//********************************Action case***********************************
CASE fb_mem.STS.State OF
	E_State_PackML.IDLE 			: 
		//Do nothing
	E_State_PackML.STARTING 		:
		Motor.Start();
		IF Motor.State = E_State_PackML.EXECUTE THEN
			fb_mem.STS.Starting_SC 		:= TRUE;	
		END_IF
	E_State_PackML.EXECUTE 			: 
		//Do nothing
	E_State_PackML.COMPLETING		:
		Motor.Stop();
		fb_mem.STS.Completing_SC := TRUE;
	E_State_PackML.COMPLETE 		:
		//Do nothing
	E_State_PackML.RESETTING 		:
		Motor.Reset();
		IF Motor.State = E_State_PackML.IDLE THEN
			fb_mem.STS.Resetting_SC 	:= TRUE;
		END_IF
	E_State_PackML.HOLDING 			:
		Motor.Stop();
		IF Motor.State = E_State_PackML.STOPPED THEN
			fb_mem.STS.Holding_SC		:= TRUE;
		END_IF
	E_State_PackML.HELD 			:
		//Do nothing
	E_State_PackML.UNHOLDING 		:
		Motor.Reset();
		Motor.Reset();
		IF Motor.State = E_State_PackML.EXECUTE THEN
			fb_mem.STS.Unholding_SC		:= TRUE;
		END_IF
	E_State_PackML.SUSPENDING 		:
		Motor.Stop();
		IF Motor.State = E_State_PackML.STOPPED THEN
			fb_mem.STS.Suspending_SC 	:= TRUE;
		END_IF
	E_State_PackML.SUSPENDED 		:
		//Do nothing
	E_State_PackML.UNSUSPENDING 	:
		Motor.Reset();
		Motor.Reset();
		IF Motor.State = E_State_PackML.EXECUTE THEN
			fb_mem.CS.Unsuspend 		:= TRUE;
		END_IF
	E_State_PackML.ABORTING			:
		Motor.Abort();
		IF Motor.State = E_State_PackML.ABORTED THEN
			fb_mem.STS.Aborting_SC 		:= TRUE;
		END_IF
	E_State_PackML.ABORTED			:		
		//Do nothing
	E_State_PackML.CLEARING 		:
		Motor.Clear();
		IF Motor.State = E_State_PackML.STOPPED THEN
			fb_mem.STS.Clearing_SC 		:= TRUE;
		END_IF
	E_State_PackML.STOPPING 		:
		IF Motor.State = E_State_PackML.STOPPED THEN
			fb_mem.STS.Stopping_SC 		:= TRUE;
		END_IF
	E_State_PackML.STOPPED 			:
		//Do nothing
END_CASE

//********************************HMI_Connection***********************************
fb_mem.STS.StringState     := TO_STRING(fb_mem.STS.State); 

//********************************ZEROING***********************************

fb_mem.CS.Auto            := FALSE;
fb_mem.CS.Manueel         := FALSE;
fb_mem.CS.Start           := FALSE;
fb_mem.CS.Stop            := FALSE;
fb_mem.CS.Reset           := FALSE;
fb_mem.CS.Abort           := FALSE;
fb_mem.CS.Clear           := FALSE;
fb_mem.CS.UnSuspend       := FALSE;
fb_mem.CS.Suspend         := FALSE;
fb_mem.CS.UnHold          := FALSE;
fb_mem.CS.Hold            := FALSE;

{warning 'add method implementation '}
METHOD Abort : BOOL
fb_mem.CS.Abort := TRUE;
END_METHOD

METHOD Aborting_SC : BOOL
VAR_INPUT
END_VAR
fb_mem.STS.Aborting_SC := TRUE;
END_METHOD

{warning 'add method implementation '}
METHOD Auto : BOOL
fb_mem.CS.Auto := TRUE;
Auto := fb_mem.STS.Auto;
END_METHOD

{warning 'add method implementation '}
METHOD Clear : BOOL
fb_mem.CS.Clear := TRUE;
END_METHOD

METHOD Clearing_SC : BOOL
VAR_INPUT
END_VAR
fb_mem.STS.Clearing_SC := TRUE;
END_METHOD

METHOD Completing_SC : BOOL
VAR_INPUT
END_VAR
fb_mem.STS.Completing_SC := TRUE;
END_METHOD

METHOD Execute_SC : BOOL
VAR_INPUT
END_VAR
fb_mem.STS.Execute_SC := TRUE;
END_METHOD

{warning 'add method implementation '}
METHOD FB_init : BOOL
VAR_INPUT
	(* if TRUE, the retain variables are initialized (warm start / cold start)*)
	bInitRetains	: BOOL;
	(* if TRUE, the instance afterwards gets moved into the copy code (online change)*)
	bInCopyCode	: BOOL;
END_VAR
END_METHOD

{warning 'add method implementation '}
METHOD Hold : BOOL
fb_mem.CS.Hold := TRUE;
END_METHOD

METHOD Holding_SC : BOOL
VAR_INPUT
END_VAR
fb_mem.STS.Holding_SC := TRUE;
END_METHOD

{warning 'add method implementation '}
METHOD Manueel : BOOL
fb_mem.CS.Manueel := TRUE;
Manueel := fb_mem.STS.Manueel;
END_METHOD

{warning 'add method implementation '}
METHOD Reset : BOOL
fb_mem.CS.Reset := TRUE;
END_METHOD

METHOD Resetting_SC : BOOL
VAR_INPUT
END_VAR
fb_mem.STS.Resetting_SC := TRUE;
END_METHOD

{warning 'add property implementation'}
PROPERTY RPM : INT
GET
END_GET
SET
END_SET
END_PROPERTY

{warning 'add method implementation '}
METHOD Start : BOOL
fb_mem.CS.Start := TRUE;
END_METHOD

METHOD Starting_SC : BOOL
VAR_INPUT
END_VAR
fb_mem.STS.Starting_SC := TRUE;
END_METHOD

{warning 'add property implementation'}
PROPERTY State : E_State_PackML
GET
State := fb_mem.STS.State;
END_GET
END_PROPERTY

{warning 'add method implementation '}
METHOD Stop : BOOL
fb_mem.CS.Stop := TRUE;
END_METHOD

METHOD Stopping_SC : BOOL
VAR_INPUT
END_VAR
fb_mem.STS.Stopping_SC := TRUE;
END_METHOD

{warning 'add method implementation '}
METHOD Suspend : BOOL
fb_mem.CS.Suspend := TRUE;
END_METHOD

METHOD Suspending_SC : BOOL
VAR_INPUT
END_VAR
fb_mem.STS.Suspending_SC := TRUE;
END_METHOD

{warning 'add property implementation'}
PROPERTY Tag : STRING
GET
Tag := fb_mem.STS.Tag;
END_GET
END_PROPERTY

{warning 'add method implementation '}
METHOD Unhold : BOOL
fb_mem.CS.Unhold := TRUE;
END_METHOD

METHOD Unholding_SC : BOOL
VAR_INPUT
END_VAR
fb_mem.STS.Unholding_SC := TRUE;
END_METHOD

{warning 'add method implementation '}
METHOD Unsuspend : BOOL
fb_mem.CS.Unsuspend := TRUE;
END_METHOD

METHOD Unsuspending_SC : BOOL
VAR_INPUT
END_VAR
fb_mem.STS.Unsuspending_SC := TRUE;
END_METHOD

{warning 'add method implementation '}
METHOD ZeroAllVar : BOOL
END_METHOD

END_FUNCTION_BLOCK

// ---- POUs/1. Control Modules/1. CM_Motor/CM_Motor.TcPOU
FUNCTION_BLOCK CM_Motor IMPLEMENTS  ITF_Motor
VAR
	fb_mem : STRUCT_CM_Motor;
END_VAR

(*
$$$$$$$$\                                                                   $$\       $$$$$$$$\                     $$\                                         $$\                     
$$  _____|                                                                  $$ |      $$  _____|                    \__|                                        \__|                    
$$ |   $$$$$$\   $$$$$$\  $$$$$$$\  $$\  $$\  $$\  $$$$$$\   $$$$$$\   $$$$$$$ |      $$ |      $$$$$$$\   $$$$$$\  $$\ $$$$$$$\   $$$$$$\   $$$$$$\   $$$$$$\  $$\ $$$$$$$\   $$$$$$\  
$$$$$\ \____$$\ $$  __$$\ $$  __$$\ $$ | $$ | $$ |$$  __$$\ $$  __$$\ $$  __$$ |      $$$$$\    $$  __$$\ $$  __$$\ $$ |$$  __$$\ $$  __$$\ $$  __$$\ $$  __$$\ $$ |$$  __$$\ $$  __$$\ 
$$  __|$$$$$$$ |$$ |  \__|$$ |  $$ |$$ | $$ | $$ |$$ /  $$ |$$ /  $$ |$$ /  $$ |      $$  __|   $$ |  $$ |$$ /  $$ |$$ |$$ |  $$ |$$$$$$$$ |$$$$$$$$ |$$ |  \__|$$ |$$ |  $$ |$$ /  $$ |
$$ |  $$  __$$ |$$ |      $$ |  $$ |$$ | $$ | $$ |$$ |  $$ |$$ |  $$ |$$ |  $$ |      $$ |      $$ |  $$ |$$ |  $$ |$$ |$$ |  $$ |$$   ____|$$   ____|$$ |      $$ |$$ |  $$ |$$ |  $$ |
$$ |  \$$$$$$$ |$$ |      $$ |  $$ |\$$$$$\$$$$  |\$$$$$$  |\$$$$$$  |\$$$$$$$ |      $$$$$$$$\ $$ |  $$ |\$$$$$$$ |$$ |$$ |  $$ |\$$$$$$$\ \$$$$$$$\ $$ |      $$ |$$ |  $$ |\$$$$$$$ |
\__|   \_______|\__|      \__|  \__| \_____\____/  \______/  \______/  \_______|      \________|\__|  \__| \____$$ |\__|\__|  \__| \_______| \_______|\__|      \__|\__|  \__| \____$$ |
                                                                                                          $$\   $$ |                                                          $$\   $$ |
      			                                                                                          \$$$$$$  |                                                          \$$$$$$  |
                                                                                                           \______/                                                            \______/ 
*)
fb_mem.STS.State := PackML_StateMachine(State			:= fb_mem.STS.State,
										Start           := fb_mem.CS.Start,
										Stop            := fb_mem.CS.Stop,
										Reset           := fb_mem.CS.Reset,
										Abort           := fb_mem.CS.Abort,
										Clear           := fb_mem.CS.Clear,
										UnSuspend       := fb_mem.CS.UnSuspend,
										Suspend         := fb_mem.CS.Suspend,
										UnHold          := fb_mem.CS.UnHold,
										Hold            := fb_mem.CS.Hold,
										Starting_SC     := fb_mem.STS.Starting_SC,
										Execute_SC      := fb_mem.STS.Execute_SC,
										Completing_SC	:= fb_mem.STS.Completing_SC,
										Resetting_SC    := fb_mem.STS.Resetting_SC,
										Holding_SC      := fb_mem.STS.Holding_SC,
										Unholding_SC    := fb_mem.STS.Unholding_SC,
										Suspending_SC   := fb_mem.STS.Suspending_SC,
										Unsuspending_SC := fb_mem.STS.Unsuspending_SC,
										Aborting_SC     := fb_mem.STS.Aborting_SC,
										Clearing_SC     := fb_mem.STS.Clearing_SC,
										Stopping_SC     := fb_mem.STS.Stopping_SC);

//********************************Auto manual logic***********************************
IF fb_mem.CS.Auto OR fb_mem.HMI.Auto THEN
	fb_mem.STS.Auto := TRUE;
	fb_mem.STS.Manueel := FALSE;
END_IF

IF fb_mem.CS.Manueel OR fb_mem.HMI.Manueel THEN
	fb_mem.STS.Auto := FALSE;
	fb_mem.STS.Manueel := TRUE;
END_IF

//********************************Toerental***********************************

fb_mem.STS.Toerental := fb_mem.CS.Toerental;

//********************************Exeptionhandling***********************************

//********************************Action case***********************************
CASE fb_mem.STS.State OF
	E_State_PackML.IDLE 			:
		//Do nothing
	E_State_PackML.STARTING 		:
		fb_mem.STS.Starting_SC 		:= TRUE;
	E_State_PackML.EXECUTE 			: 
		//Do nothing
	E_State_PackML.COMPLETING		:
		fb_mem.STS.Completing_SC := TRUE;
	E_State_PackML.COMPLETE 		:
		IF fb_mem.CS.Clear AND fb_mem.STS.Auto OR fb_mem.HMI.Clear AND fb_mem.STS.Manueel THEN
			fb_mem.STS.Completing_SC := TRUE;
		END_IF
	E_State_PackML.RESETTING 		:
		FB_init(0,0);
		fb_mem.STS.Resetting_SC 	:= TRUE;
	E_State_PackML.HOLDING 			:
		fb_mem.STS.Unholding_SC		:= TRUE;
	E_State_PackML.HELD 			:
		//Do nothing
	E_State_PackML.UNHOLDING 		:
		fb_mem.STS.Unholding_SC		:= TRUE;
	E_State_PackML.SUSPENDING 		:
		fb_mem.STS.Suspending_SC 	:= TRUE;
	E_State_PackML.SUSPENDED 		:
		fb_mem.CS.Unsuspend 		:= TRUE;
	E_State_PackML.UNSUSPENDING 	:
		fb_mem.STS.Unsuspending_SC 	:= TRUE;
	E_State_PackML.ABORTED			:
		//Do nothing
	E_State_PackML.ABORTING			:
		fb_mem.STS.Aborting_SC 		:= TRUE;
	E_State_PackML.CLEARING 		:
		fb_mem.STS.Clearing_SC 		:= TRUE;
	E_State_PackML.STOPPING 		:
		fb_mem.STS.Stopping_SC 		:= TRUE;
	E_State_PackML.STOPPED 			:
		//Do nothing
		
END_CASE




//Zero all CS signals
fb_mem.CS.Auto			:= FALSE;
fb_mem.CS.Manueel 		:= FALSE;
fb_mem.CS.Abort			:= FALSE;
fb_mem.CS.Reset			:= FALSE;
fb_mem.CS.Richting_L	:= FALSE;
fb_mem.CS.Richting_R	:= FALSE;
fb_mem.CS.Start			:= FALSE;
fb_mem.CS.Stop			:= FALSE;

//Zero all HMI signals
fb_mem.HMI.Auto			:= FALSE;
fb_mem.HMI.Manueel 		:= FALSE;
fb_mem.HMI.Abort		:= FALSE;
fb_mem.HMI.Reset		:= FALSE;
fb_mem.HMI.Richting_L	:= FALSE;
fb_mem.HMI.Richting_R	:= FALSE;
fb_mem.HMI.Start		:= FALSE;
fb_mem.HMI.Stop			:= FALSE;

{warning 'add method implementation '}
METHOD Abort : BOOL
fb_mem.CS.Abort := TRUE;

Abort := fb_mem.CS.Abort;
END_METHOD

PROPERTY Auto : BOOl
GET
AUTO := fb_mem.STS.Auto;
END_GET
SET
fb_mem.CS.Auto := AUTO;
END_SET
END_PROPERTY

METHOD Clear : BOOL
VAR_INPUT
END_VAR
fb_mem.CS.Clear := TRUE;

Clear := fb_mem.CS.Abort;
END_METHOD

{warning 'add property implementation'}
PROPERTY Error_State : E_Motor_Error_State
GET
Error_State := fb_mem.STS.Error_State;
END_GET
END_PROPERTY

METHOD FB_init : BOOL
VAR_INPUT
	bInitRetains : BOOL; // if TRUE, the retain variables are initialized (warm start / cold start)
	bInCopyCode : BOOL;  // if TRUE, the instance afterwards gets moved into the copy code (online change)
END_VAR
fb_mem.STS.State := E_State_PackML.IDLE;
END_METHOD

PROPERTY Manueel : BOOl
GET
Manueel := fb_mem.STS.Manueel;
END_GET
SET
fb_mem.CS.Manueel :=  Manueel;
END_SET
END_PROPERTY

{warning 'add method implementation '}
METHOD Reset : BOOL
fb_mem.CS.Reset := TRUE;

Reset := fb_mem.CS.Reset;
END_METHOD

{warning 'add property implementation'}
PROPERTY Richting_L : BOOL
GET
Richting_L := fb_mem.STS.Richting_L;
END_GET
SET
fb_mem.CS.Richting_L := Richting_L;
END_SET
END_PROPERTY

{warning 'add property implementation'}
PROPERTY Richting_R : BOOL
GET
Richting_R := fb_mem.STS.Richting_R;
END_GET
SET
fb_mem.CS.Richting_R := Richting_R;
END_SET
END_PROPERTY

{warning 'add method implementation '}
METHOD Start : BOOL
fb_mem.CS.Start := TRUE;

Start := fb_mem.CS.Start;
END_METHOD

{warning 'add property implementation'}
PROPERTY State : E_Motor_State
GET
END_GET
END_PROPERTY

{warning 'add method implementation '}
METHOD Stop : BOOL
fb_mem.CS.Stop := TRUE;

Stop := fb_mem.CS.Stop;
END_METHOD

PROPERTY Tag : STRING
GET
Tag := fb_mem.STS.Tag;
END_GET
END_PROPERTY

{warning 'add method implementation '}
METHOD Toerental : INT
fb_mem.CS.Toerental := Toerental;

Toerental := fb_mem.STS.Toerental;
END_METHOD

END_FUNCTION_BLOCK

// ---- POUs/4. Management/3. PackML/PackML_StateMachine.TcPOU
FUNCTION PackML_StateMachine : E_State_PackML
VAR_INPUT
	State		: E_State_PackML;
	Start		: BOOL;
	Stop		: BOOL;
	Reset		: BOOL;
	Abort		: BOOL;
	Clear		: BOOL;
	UnSuspend	: BOOL;
	Suspend		: BOOL;
	UnHold		: BOOL;
	Hold		: BOOL;
	
	Starting_SC 	: BOOL;
	Execute_SC 		: BOOL;
	Resetting_SC 	: BOOL;
	Holding_SC 		: BOOL;
	Unholding_SC 	: BOOL;
	Suspending_SC	: BOOL;
	Unsuspending_SC	: BOOL;
	Aborting_SC		: BOOL;
	Clearing_SC		: BOOL;
	Completing_SC	: BOOL;
	Stopping_SC		: BOOL;
END_VAR
VAR
	bFirstCylceBit	: BOOL := TRUE;
END_VAR

(*
$$$$$$$$\                                                                   $$\       $$$$$$$$\                     $$\                                         $$\                     
$$  _____|                                                                  $$ |      $$  _____|                    \__|                                        \__|                    
$$ |   $$$$$$\   $$$$$$\  $$$$$$$\  $$\  $$\  $$\  $$$$$$\   $$$$$$\   $$$$$$$ |      $$ |      $$$$$$$\   $$$$$$\  $$\ $$$$$$$\   $$$$$$\   $$$$$$\   $$$$$$\  $$\ $$$$$$$\   $$$$$$\  
$$$$$\ \____$$\ $$  __$$\ $$  __$$\ $$ | $$ | $$ |$$  __$$\ $$  __$$\ $$  __$$ |      $$$$$\    $$  __$$\ $$  __$$\ $$ |$$  __$$\ $$  __$$\ $$  __$$\ $$  __$$\ $$ |$$  __$$\ $$  __$$\ 
$$  __|$$$$$$$ |$$ |  \__|$$ |  $$ |$$ | $$ | $$ |$$ /  $$ |$$ /  $$ |$$ /  $$ |      $$  __|   $$ |  $$ |$$ /  $$ |$$ |$$ |  $$ |$$$$$$$$ |$$$$$$$$ |$$ |  \__|$$ |$$ |  $$ |$$ /  $$ |
$$ |  $$  __$$ |$$ |      $$ |  $$ |$$ | $$ | $$ |$$ |  $$ |$$ |  $$ |$$ |  $$ |      $$ |      $$ |  $$ |$$ |  $$ |$$ |$$ |  $$ |$$   ____|$$   ____|$$ |      $$ |$$ |  $$ |$$ |  $$ |
$$ |  \$$$$$$$ |$$ |      $$ |  $$ |\$$$$$\$$$$  |\$$$$$$  |\$$$$$$  |\$$$$$$$ |      $$$$$$$$\ $$ |  $$ |\$$$$$$$ |$$ |$$ |  $$ |\$$$$$$$\ \$$$$$$$\ $$ |      $$ |$$ |  $$ |\$$$$$$$ |
\__|   \_______|\__|      \__|  \__| \_____\____/  \______/  \______/  \_______|      \________|\__|  \__| \____$$ |\__|\__|  \__| \_______| \_______|\__|      \__|\__|  \__| \____$$ |
                                                                                                          $$\   $$ |                                                          $$\   $$ |
                                                                                                          \$$$$$$  |                                                          \$$$$$$  |
                                                                                                           \______/                                                            \______/ 
*)
CASE State OF
	E_State_PackML.IDLE 			:
		//HAPPY FLOW		
		IF Start AND NOT Abort THEN
			State := E_State_PackML.STARTING;
		END_IF
		
		//EXEPTION HANDLING
		IF Abort THEN
			State:= E_State_PackML.ABORTING;
		END_IF
		IF Stop THEN
			State:= E_State_PackML.STOPPING;
		END_IF
	
	E_State_PackML.STARTING 		:
		//HAPPY FLOW		
		IF Starting_SC AND NOT Abort THEN
			State:= E_State_PackML.EXECUTE;
		END_IF
		
		//EXEPTION HANDLING
		IF Abort THEN
			State:= E_State_PackML.ABORTING;
		END_IF
		IF Stop THEN
			State:= E_State_PackML.STOPPING;
		END_IF
	
	E_State_PackML.EXECUTE 			:
		//HAPPY FLOW		
		IF Execute_SC AND NOT Abort THEN
			State := E_State_PackML.COMPLETING;
		END_IF
		
		IF Hold THEN
			State := E_State_PackML.HOLDING;
		END_IF
		
		IF Suspend THEN
			State := E_State_PackML.SUSPENDING;
		END_IF
		
		//EXEPTION HANDLING
		IF Abort THEN
			State:= E_State_PackML.ABORTING;
		END_IF
		IF Stop THEN
			State:= E_State_PackML.STOPPING;
		END_IF
	E_State_PackML.COMPLETING		:
		//HAPPY FLOW
		IF Completing_SC THEN
			State := E_State_PackML.COMPLETE;
		END_IF
		//EXEPTION HANDLING
		IF Abort THEN
			State := E_State_PackML.ABORTING;
		END_IF
		IF Stop	THEN
			State := E_State_PackML.STOPPING;
		END_IF
	E_State_PackML.COMPLETE 		:
		//HAPPY FLOW
		IF Reset AND NOT ABORT THEN
			State:= E_State_PackML.RESETTING;
		END_IF
		//EXEPTION HANDLING
		IF Abort THEN
			State := E_State_PackML.ABORTING;
		END_IF
		IF Stop	THEN
			State := E_State_PackML.STOPPING;
		END_IF
	
	E_State_PackML.RESETTING 		:
		//HAPPY FLOW		
		IF Resetting_SC AND NOT Abort THEN
			State:= E_State_PackML.IDLE;
		END_IF
		
		//EXEPTION HANDLING
		IF Abort THEN
			State:= E_State_PackML.ABORTING;
		END_IF
		IF Stop THEN
			State:= E_State_PackML.STOPPING;
		END_IF
	
	E_State_PackML.HOLDING 			:
		//HAPPY FLOW		
		IF Holding_SC AND NOT Abort THEN
			State:= E_State_PackML.HELD;
		END_IF
		
		//EXEPTION HANDLING
		IF Abort THEN
			State:= E_State_PackML.ABORTING;
		END_IF
		IF Stop THEN
			State:= E_State_PackML.STOPPING;
		END_IF
		
	
	E_State_PackML.HELD 			:
		//HAPPY FLOW		
		IF Unhold AND NOT Abort THEN
			State := E_State_PackML.UNHOLDING;
		END_IF
		
		//EXEPTION HANDLING
		IF Abort THEN
			State:= E_State_PackML.ABORTING;
		END_IF
		IF Stop THEN
			State:= E_State_PackML.STOPPING;
		END_IF
	
	E_State_PackML.UNHOLDING 		:
		//HAPPY FLOW		
		IF Unholding_SC AND NOT Abort THEN
			State:= E_State_PackML.EXECUTE;
		END_IF
		
		//EXEPTION HANDLING
		IF Abort THEN
			State:= E_State_PackML.ABORTING;
		END_IF
		IF Stop THEN
			State:= E_State_PackML.STOPPING;
		END_IF
	
	E_State_PackML.SUSPENDING 		:
		//HAPPY FLOW		
		IF Suspending_SC AND NOT Abort THEN
			State:= E_State_PackML.SUSPENDED;
		END_IF
		
		//EXEPTION HANDLING
		IF Abort THEN
			State:= E_State_PackML.ABORTING;
		END_IF
		IF Stop THEN
			State:= E_State_PackML.STOPPING;
		END_IF
	
	
	E_State_PackML.SUSPENDED 		:
		//HAPPY FLOW		
		IF Unsuspend AND NOT Abort THEN
			State:= E_State_PackML.UNSUSPENDING;
		END_IF
		
		//EXEPTION HANDLING
		IF Abort THEN
			State:= E_State_PackML.ABORTING;
		END_IF
		IF Stop THEN
			State:= E_State_PackML.STOPPING;
		END_IF
	
	E_State_PackML.UNSUSPENDING 	:
		//HAPPY FLOW		
		IF Unsuspending_SC AND NOT Abort THEN
			State:= E_State_PackML.EXECUTE;
		END_IF
		
		//EXEPTION HANDLING
		IF Abort THEN
			State:= E_State_PackML.ABORTING;
		END_IF
		IF Stop THEN
			State:= E_State_PackML.STOPPING;
		END_IF
	
	E_State_PackML.ABORTED			:
		//HAPPY FLOW		
		IF Clear THEN
			State:= E_State_PackML.CLEARING;
		END_IF
	
		
	E_State_PackML.ABORTING			:
		//HAPPY FLOW		
		IF Aborting_SC THEN
			State:= E_State_PackML.ABORTED;
		END_IF
	
		
	E_State_PackML.CLEARING 		:
		//HAPPY FLOW		
		IF Clearing_SC THEN
			State:= E_State_PackML.STOPPED;
		END_IF
		
		//EXEPTION HANDLING
		IF Abort THEN
			State:= E_State_PackML.ABORTING;
		END_IF
		
		
	E_State_PackML.STOPPING 		:
		//HAPPY FLOW
		IF Stopping_SC THEN
			State:= E_State_PackML.STOPPED;
		END_IF
		
		//EXEPTION HANDLING
		IF Abort THEN
			State:= E_State_PackML.ABORTING;
		END_IF
		
	
	E_State_PackML.STOPPED 			: 
		//HAPPY FLOW
		IF Reset AND NOT Abort THEN
			State := E_State_PackML.RESETTING;
		END_IF
		
		//EXEPTION HANDLING
		IF Abort THEN
			State:= E_State_PackML.ABORTING;
		END_IF
END_CASE

PackML_StateMachine := State;

END_FUNCTION

// ---- POUs/1. Control Modules/2. CM_Sensor/CM_Sensor.TcPOU
FUNCTION_BLOCK CM_Sensor IMPLEMENTS  ITF_Sensor
VAR
	fb_mem : STRUCT_CM_Sensor;
END_VAR

(*
$$$$$$$$\                                                                   $$\       $$$$$$$$\                     $$\                                         $$\                     
$$  _____|                                                                  $$ |      $$  _____|                    \__|                                        \__|                    
$$ |   $$$$$$\   $$$$$$\  $$$$$$$\  $$\  $$\  $$\  $$$$$$\   $$$$$$\   $$$$$$$ |      $$ |      $$$$$$$\   $$$$$$\  $$\ $$$$$$$\   $$$$$$\   $$$$$$\   $$$$$$\  $$\ $$$$$$$\   $$$$$$\  
$$$$$\ \____$$\ $$  __$$\ $$  __$$\ $$ | $$ | $$ |$$  __$$\ $$  __$$\ $$  __$$ |      $$$$$\    $$  __$$\ $$  __$$\ $$ |$$  __$$\ $$  __$$\ $$  __$$\ $$  __$$\ $$ |$$  __$$\ $$  __$$\ 
$$  __|$$$$$$$ |$$ |  \__|$$ |  $$ |$$ | $$ | $$ |$$ /  $$ |$$ /  $$ |$$ /  $$ |      $$  __|   $$ |  $$ |$$ /  $$ |$$ |$$ |  $$ |$$$$$$$$ |$$$$$$$$ |$$ |  \__|$$ |$$ |  $$ |$$ /  $$ |
$$ |  $$  __$$ |$$ |      $$ |  $$ |$$ | $$ | $$ |$$ |  $$ |$$ |  $$ |$$ |  $$ |      $$ |      $$ |  $$ |$$ |  $$ |$$ |$$ |  $$ |$$   ____|$$   ____|$$ |      $$ |$$ |  $$ |$$ |  $$ |
$$ |  \$$$$$$$ |$$ |      $$ |  $$ |\$$$$$\$$$$  |\$$$$$$  |\$$$$$$  |\$$$$$$$ |      $$$$$$$$\ $$ |  $$ |\$$$$$$$ |$$ |$$ |  $$ |\$$$$$$$\ \$$$$$$$\ $$ |      $$ |$$ |  $$ |\$$$$$$$ |
\__|   \_______|\__|      \__|  \__| \_____\____/  \______/  \______/  \_______|      \________|\__|  \__| \____$$ |\__|\__|  \__| \_______| \_______|\__|      \__|\__|  \__| \____$$ |
                                                                                                          $$\   $$ |                                                          $$\   $$ |
                                                                                                          \$$$$$$  |                                                          \$$$$$$  |
                                                                                                           \______/                                                            \______/ 
*)

fb_mem.STS.Output := fb_mem.CS.Output;

//Zero all CS signals
fb_mem.CS.Auto		:= FALSE;
fb_mem.CS.Manueel 	:= FALSE;
fb_mem.CS.Output	:= FALSE;

//Zero all HMI signals
fb_mem.HMI.Auto		:= FALSE;
fb_mem.HMI.Manueel 	:= FALSE;
fb_mem.HMI.Output	:= FALSE;

PROPERTY Auto : BOOl
GET
AUTO := fb_mem.STS.Auto;
END_GET
SET
fb_mem.CS.Auto := AUTO;
END_SET
END_PROPERTY

METHOD FB_init : BOOL
VAR_INPUT
	bInitRetains : BOOL; // if TRUE, the retain variables are initialized (warm start / cold start)
	bInCopyCode : BOOL;  // if TRUE, the instance afterwards gets moved into the copy code (online change)
END_VAR
fb_mem.STS.Output := FALSE;
END_METHOD

PROPERTY Manueel : BOOl
GET
Manueel := fb_mem.STS.Manueel;
END_GET
SET
fb_mem.CS.Manueel :=  Manueel;
END_SET
END_PROPERTY

PROPERTY Output : BOOl
GET
Output := fb_mem.STS.Output;
END_GET
SET
fb_mem.CS.Output := Output;
END_SET
END_PROPERTY

PROPERTY Tag : STRING
GET
Tag := fb_mem.STS.Tag;
END_GET
END_PROPERTY

END_FUNCTION_BLOCK

// ---- POUs/1. Control Modules/4. CM_Valve/CM_Valve.TcPOU
FUNCTION_BLOCK CM_Valve IMPLEMENTS  ITF_Valve2
VAR
	fb_mem : STRUCT_CM_Valve;
END_VAR

(*
$$$$$$$$\                                                                   $$\       $$$$$$$$\                     $$\                                         $$\                     
$$  _____|                                                                  $$ |      $$  _____|                    \__|                                        \__|                    
$$ |   $$$$$$\   $$$$$$\  $$$$$$$\  $$\  $$\  $$\  $$$$$$\   $$$$$$\   $$$$$$$ |      $$ |      $$$$$$$\   $$$$$$\  $$\ $$$$$$$\   $$$$$$\   $$$$$$\   $$$$$$\  $$\ $$$$$$$\   $$$$$$\  
$$$$$\ \____$$\ $$  __$$\ $$  __$$\ $$ | $$ | $$ |$$  __$$\ $$  __$$\ $$  __$$ |      $$$$$\    $$  __$$\ $$  __$$\ $$ |$$  __$$\ $$  __$$\ $$  __$$\ $$  __$$\ $$ |$$  __$$\ $$  __$$\ 
$$  __|$$$$$$$ |$$ |  \__|$$ |  $$ |$$ | $$ | $$ |$$ /  $$ |$$ /  $$ |$$ /  $$ |      $$  __|   $$ |  $$ |$$ /  $$ |$$ |$$ |  $$ |$$$$$$$$ |$$$$$$$$ |$$ |  \__|$$ |$$ |  $$ |$$ /  $$ |
$$ |  $$  __$$ |$$ |      $$ |  $$ |$$ | $$ | $$ |$$ |  $$ |$$ |  $$ |$$ |  $$ |      $$ |      $$ |  $$ |$$ |  $$ |$$ |$$ |  $$ |$$   ____|$$   ____|$$ |      $$ |$$ |  $$ |$$ |  $$ |
$$ |  \$$$$$$$ |$$ |      $$ |  $$ |\$$$$$\$$$$  |\$$$$$$  |\$$$$$$  |\$$$$$$$ |      $$$$$$$$\ $$ |  $$ |\$$$$$$$ |$$ |$$ |  $$ |\$$$$$$$\ \$$$$$$$\ $$ |      $$ |$$ |  $$ |\$$$$$$$ |
\__|   \_______|\__|      \__|  \__| \_____\____/  \______/  \______/  \_______|      \________|\__|  \__| \____$$ |\__|\__|  \__| \_______| \_______|\__|      \__|\__|  \__| \____$$ |
                                                                                                          $$\   $$ |                                                          $$\   $$ |
      			                                                                                          \$$$$$$  |                                                          \$$$$$$  |
                                                                                                           \______/                                                            \______/ 
*)
fb_mem.STS.State := PackML_StateMachine(State			:= fb_mem.STS.State,
										Start           := fb_mem.CS.Start,
										Stop            := fb_mem.CS.Stop,
										Reset           := fb_mem.CS.Reset,
										Abort           := fb_mem.CS.Abort,
										Clear           := fb_mem.CS.Clear,
										UnSuspend       := fb_mem.CS.UnSuspend,
										Suspend         := fb_mem.CS.Suspend,
										UnHold          := fb_mem.CS.UnHold,
										Hold            := fb_mem.CS.Hold,
										Starting_SC     := fb_mem.STS.Starting_SC,
										Execute_SC      := fb_mem.STS.Execute_SC,
										Completing_SC	:= fb_mem.STS.Completing_SC,
										Resetting_SC    := fb_mem.STS.Resetting_SC,
										Holding_SC      := fb_mem.STS.Holding_SC,
										Unholding_SC    := fb_mem.STS.Unholding_SC,
										Suspending_SC   := fb_mem.STS.Suspending_SC,
										Unsuspending_SC := fb_mem.STS.Unsuspending_SC,
										Aborting_SC     := fb_mem.STS.Aborting_SC,
										Clearing_SC     := fb_mem.STS.Clearing_SC,
										Stopping_SC     := fb_mem.STS.Stopping_SC);

//********************************Auto manual logic***********************************
IF fb_mem.CS.Auto OR fb_mem.HMI.Auto THEN
	fb_mem.STS.Auto := TRUE;
	fb_mem.STS.Manueel := FALSE;
END_IF

IF fb_mem.CS.Manueel OR fb_mem.HMI.Manueel THEN
	fb_mem.STS.Auto := FALSE;
	fb_mem.STS.Manueel := TRUE;
END_IF

//********************************Exeptionhandling***********************************

//********************************Action case***********************************
CASE fb_mem.STS.State OF
	E_State_PackML.IDLE 			:
		//Do nothing
	E_State_PackML.STARTING 		:
		fb_mem.STS.Starting_SC 		:= TRUE;
	E_State_PackML.EXECUTE 			: 
		//Do nothing
	E_State_PackML.COMPLETING		:
		fb_mem.STS.Completing_SC := TRUE;
	E_State_PackML.COMPLETE 		:
		IF fb_mem.CS.Clear AND fb_mem.STS.Auto OR fb_mem.HMI.Clear AND fb_mem.STS.Manueel THEN
			fb_mem.STS.Completing_SC := TRUE;
		END_IF
	E_State_PackML.RESETTING 		:
		FB_init(0,0);
		fb_mem.STS.Resetting_SC 	:= TRUE;
	E_State_PackML.HOLDING 			:
		fb_mem.STS.Unholding_SC		:= TRUE;
	E_State_PackML.HELD 			:
		//Do nothing
	E_State_PackML.UNHOLDING 		:
		fb_mem.STS.Unholding_SC		:= TRUE;
	E_State_PackML.SUSPENDING 		:
		fb_mem.STS.Suspending_SC 	:= TRUE;
	E_State_PackML.SUSPENDED 		:
		fb_mem.CS.Unsuspend 		:= TRUE;
	E_State_PackML.UNSUSPENDING 	:
		fb_mem.STS.Unsuspending_SC 	:= TRUE;
	E_State_PackML.ABORTED			:
		//Do nothing
	E_State_PackML.ABORTING			:
		fb_mem.STS.Aborting_SC 		:= TRUE;
	E_State_PackML.CLEARING 		:
		fb_mem.STS.Clearing_SC 		:= TRUE;
	E_State_PackML.STOPPING 		:
		fb_mem.STS.Stopping_SC 		:= TRUE;
	E_State_PackML.STOPPED 			:
		//Do nothing
		
END_CASE




//Zero all CS signals
fb_mem.CS.Auto			:= FALSE;
fb_mem.CS.Manueel 		:= FALSE;
fb_mem.CS.Abort			:= FALSE;
fb_mem.CS.Reset			:= FALSE;
fb_mem.CS.Start			:= FALSE;
fb_mem.CS.Stop			:= FALSE;

//Zero all HMI signals
fb_mem.HMI.Auto			:= FALSE;
fb_mem.HMI.Manueel 		:= FALSE;
fb_mem.HMI.Abort		:= FALSE;
fb_mem.HMI.Reset		:= FALSE;
fb_mem.HMI.Start		:= FALSE;
fb_mem.HMI.Stop			:= FALSE;

{warning 'add method implementation '}
METHOD Abort : BOOL
fb_mem.CS.Abort := TRUE;

Abort := fb_mem.CS.Abort;
END_METHOD

PROPERTY Auto : BOOl
GET
AUTO := fb_mem.STS.Auto;
END_GET
SET
fb_mem.CS.Auto := AUTO;
END_SET
END_PROPERTY

METHOD Clear : BOOL
VAR_INPUT
END_VAR
fb_mem.CS.Clear := TRUE;

Clear := fb_mem.CS.Abort;
END_METHOD

{warning 'add method implementation '}
METHOD Close : BOOL
fb_mem.CS.Close := TRUE;
fb_mem.STS.Close:=TRUE;
fb_mem.STS.Open:=FALSE;
Close := fb_mem.STS.Close;
END_METHOD

{warning 'add property implementation'}
PROPERTY Error_State : E_Motor_Error_State
GET
Error_State := fb_mem.STS.Error_State;
END_GET
END_PROPERTY

METHOD FB_init : BOOL
VAR_INPUT
	bInitRetains : BOOL; // if TRUE, the retain variables are initialized (warm start / cold start)
	bInCopyCode : BOOL;  // if TRUE, the instance afterwards gets moved into the copy code (online change)
END_VAR
fb_mem.STS.State := E_State_PackML.IDLE;
END_METHOD

PROPERTY Manueel : BOOl
GET
Manueel := fb_mem.STS.Manueel;
END_GET
SET
fb_mem.CS.Manueel :=  Manueel;
END_SET
END_PROPERTY

{warning 'add method implementation '}
METHOD Open : BOOL
fb_mem.CS.Open := TRUE;
fb_mem.STS.Open:=TRUE;
fb_mem.STS.Close:=FALSE;
Open := fb_mem.STS.Open;
END_METHOD

{warning 'add method implementation '}
METHOD Reset : BOOL
fb_mem.CS.Reset := TRUE;

Reset := fb_mem.CS.Reset;
END_METHOD

{warning 'add method implementation '}
METHOD Start : BOOL
fb_mem.CS.Start := TRUE;

Start := fb_mem.CS.Start;
END_METHOD

{warning 'add property implementation'}
PROPERTY State : E_Motor_State
GET
END_GET
END_PROPERTY

{warning 'add method implementation '}
METHOD Stop : BOOL
fb_mem.CS.Stop := TRUE;

Stop := fb_mem.CS.Stop;
END_METHOD

PROPERTY Tag : STRING
GET
Tag := fb_mem.STS.Tag;
END_GET
END_PROPERTY

END_FUNCTION_BLOCK

// ---- POUs/2. Equipment Modules/2. EM_Filling/EM_Filling.TcPOU
FUNCTION_BLOCK EM_Filling IMPLEMENTS ITF_PackML
VAR
	fb_mem : STRUCT_EM_Filling;
	bFirstCycleExecuted : BOOL;
	
	//Submodules
	EM_FillerA1				: EM_Machine;
	EM_FillerA2				: EM_Machine;
	EM_TransportFillers		: EM_Transport;
	EM_OutfeedFillers		: EM_Transport_Mechanische_Stop;
	
	
END_VAR

(*
$$$$$$$$\                                                                   $$\       $$$$$$$$\                     $$\                                         $$\                     
$$  _____|                                                                  $$ |      $$  _____|                    \__|                                        \__|                    
$$ |   $$$$$$\   $$$$$$\  $$$$$$$\  $$\  $$\  $$\  $$$$$$\   $$$$$$\   $$$$$$$ |      $$ |      $$$$$$$\   $$$$$$\  $$\ $$$$$$$\   $$$$$$\   $$$$$$\   $$$$$$\  $$\ $$$$$$$\   $$$$$$\  
$$$$$\ \____$$\ $$  __$$\ $$  __$$\ $$ | $$ | $$ |$$  __$$\ $$  __$$\ $$  __$$ |      $$$$$\    $$  __$$\ $$  __$$\ $$ |$$  __$$\ $$  __$$\ $$  __$$\ $$  __$$\ $$ |$$  __$$\ $$  __$$\ 
$$  __|$$$$$$$ |$$ |  \__|$$ |  $$ |$$ | $$ | $$ |$$ /  $$ |$$ /  $$ |$$ /  $$ |      $$  __|   $$ |  $$ |$$ /  $$ |$$ |$$ |  $$ |$$$$$$$$ |$$$$$$$$ |$$ |  \__|$$ |$$ |  $$ |$$ /  $$ |
$$ |  $$  __$$ |$$ |      $$ |  $$ |$$ | $$ | $$ |$$ |  $$ |$$ |  $$ |$$ |  $$ |      $$ |      $$ |  $$ |$$ |  $$ |$$ |$$ |  $$ |$$   ____|$$   ____|$$ |      $$ |$$ |  $$ |$$ |  $$ |
$$ |  \$$$$$$$ |$$ |      $$ |  $$ |\$$$$$\$$$$  |\$$$$$$  |\$$$$$$  |\$$$$$$$ |      $$$$$$$$\ $$ |  $$ |\$$$$$$$ |$$ |$$ |  $$ |\$$$$$$$\ \$$$$$$$\ $$ |      $$ |$$ |  $$ |\$$$$$$$ |
\__|   \_______|\__|      \__|  \__| \_____\____/  \______/  \______/  \_______|      \________|\__|  \__| \____$$ |\__|\__|  \__| \_______| \_______|\__|      \__|\__|  \__| \____$$ |
                                                                                                          $$\   $$ |                                                          $$\   $$ |
                                                                                                          \$$$$$$  |                                                          \$$$$$$  |
                                                                                                           \______/                                                            \______/ 
*)//********************************Initiating***********************************
fb_mem.STS.State := PackML_StateMachine(State			:= fb_mem.STS.State,
										Start           := fb_mem.CS.Start,
										Stop            := fb_mem.CS.Stop,
										Reset           := fb_mem.CS.Reset,
										Abort           := fb_mem.CS.Abort,
										Clear           := fb_mem.CS.Clear,
										UnSuspend       := fb_mem.CS.UnSuspend,
										Suspend         := fb_mem.CS.Suspend,
										UnHold          := fb_mem.CS.UnHold,
										Hold            := fb_mem.CS.Hold,
										Starting_SC     := fb_mem.STS.Starting_SC,
										Execute_SC      := fb_mem.STS.Execute_SC,
										Resetting_SC    := fb_mem.STS.Resetting_SC,
										Holding_SC      := fb_mem.STS.Holding_SC,
										Unholding_SC    := fb_mem.STS.Unholding_SC,
										Suspending_SC   := fb_mem.STS.Suspending_SC,
										Unsuspending_SC := fb_mem.STS.Unsuspending_SC,
										Aborting_SC     := fb_mem.STS.Aborting_SC,
										Clearing_SC     := fb_mem.STS.Clearing_SC,
										Completing_SC	:= fb_mem.STS.Completing_SC,
										Stopping_SC     := fb_mem.STS.Stopping_SC);

//********************************Init***********************************
EM_FillerA1();
EM_FillerA2();	
EM_TransportFillers();
EM_OutfeedFillers();

IF fb_mem.STS.Starting_SC THEN
	EM_FillerA1.Starting_SC();
	EM_FillerA2.Starting_SC();
	EM_TransportFillers.Starting_SC();
	EM_OutfeedFillers.Starting_SC();
END_IF
IF fb_mem.STS.Execute_SC THEN
	EM_FillerA1.Execute_SC();
	EM_FillerA2.Execute_SC();
	EM_TransportFillers.Execute_SC();
	EM_OutfeedFillers.Execute_SC();
END_IF
IF fb_mem.STS.Resetting_SC THEN
	EM_FillerA1.Resetting_SC();
	EM_FillerA2.Resetting_SC();
	EM_TransportFillers.Resetting_SC();
	EM_OutfeedFillers.Resetting_SC();
END_IF
IF fb_mem.STS.Holding_SC THEN
	EM_FillerA1.Holding_SC();
	EM_FillerA2.Holding_SC();
	EM_TransportFillers.Holding_SC();
	EM_OutfeedFillers.Holding_SC();
END_IF
IF fb_mem.STS.Unholding_SC THEN
	EM_FillerA1.Unholding_SC();
	EM_FillerA2.Unholding_SC();
	EM_TransportFillers.Unholding_SC();
	EM_OutfeedFillers.Unholding_SC();
END_IF
IF fb_mem.STS.Suspending_SC THEN
	EM_FillerA1.Suspending_SC();
	EM_FillerA2.Suspending_SC();
	EM_TransportFillers.Suspending_SC();
	EM_OutfeedFillers.Suspending_SC();
END_IF
IF fb_mem.STS.Unsuspending_SC THEN
	EM_FillerA1.Unsuspending_SC();
	EM_FillerA2.Unsuspending_SC();
	EM_TransportFillers.Unsuspending_SC();
	EM_OutfeedFillers.Unsuspending_SC();
END_IF
IF fb_mem.STS.Aborting_SC THEN
	EM_FillerA1.Aborting_SC();
	EM_FillerA2.Aborting_SC();
	EM_TransportFillers.Aborting_SC();
	EM_OutfeedFillers.Aborting_SC();
END_IF
IF fb_mem.STS.Clearing_SC THEN
	EM_FillerA1.Clearing_SC();
	EM_FillerA2.Clearing_SC();
	EM_TransportFillers.Clearing_SC();
	EM_OutfeedFillers.Clearing_SC();
END_IF
IF fb_mem.STS.Stopping_SC THEN
	EM_FillerA1.Stopping_SC();
	EM_FillerA2.Stopping_SC();
	EM_TransportFillers.Stopping_SC();
	EM_OutfeedFillers.Stopping_SC();
END_IF
IF fb_mem.STS.Completing_SC THEN
	EM_FillerA1.Completing_SC();
	EM_FillerA2.Completing_SC();
	EM_TransportFillers.Completing_SC();
	EM_OutfeedFillers.Completing_SC();
END_IF
								
//********************************ZEROING***********************************
fb_mem.STS.Starting_SC 		:= FALSE;
fb_mem.STS.Execute_SC 		:= FALSE;
fb_mem.STS.Resetting_SC 	:= FALSE;
fb_mem.STS.Holding_SC 		:= FALSE;
fb_mem.STS.Unholding_SC 	:= FALSE;
fb_mem.STS.Suspending_SC 	:= FALSE;
fb_mem.STS.Unsuspending_SC 	:= FALSE;
fb_mem.STS.Aborting_SC 		:= FALSE;
fb_mem.STS.Clearing_SC 		:= FALSE;
fb_mem.STS.Stopping_SC 		:= FALSE;
fb_mem.STS.Completing_SC 	:= FALSE;

//********************************Auto manual logic***********************************
IF NOT bFirstCycleExecuted THEN
	EM_FillerA1.Auto();
	EM_FillerA2.Auto();
	EM_TransportFillers.Auto();
	EM_OutfeedFillers.Auto();
	bFirstCycleExecuted := TRUE;
END_IF

IF fb_mem.CS.Auto OR fb_mem.HMI.Auto THEN
	fb_mem.STS.Auto := TRUE;
	fb_mem.STS.Manueel := FALSE;
END_IF

IF fb_mem.CS.Manueel OR fb_mem.HMI.Manueel THEN
	fb_mem.STS.Auto := FALSE;
	fb_mem.STS.Manueel := TRUE;
END_IF


IF fb_mem.CS.Reset THEN
	EM_FillerA1.Reset();
	EM_FillerA2.Reset();
	EM_TransportFillers.Reset();
	EM_OutfeedFillers.Reset();
END_IF

IF fb_mem.CS.Abort THEN
	EM_FillerA1.Abort();
	EM_FillerA2.Abort();
	EM_TransportFillers.Abort();
	EM_OutfeedFillers.Abort();
END_IF

IF fb_mem.CS.Clear THEN
	EM_FillerA1.Clear();
	EM_FillerA2.Clear();
	EM_TransportFillers.Clear();
	EM_OutfeedFillers.Clear();
END_IF

IF fb_mem.CS.UnSuspend THEN
	EM_FillerA1.UnSuspend();
	EM_FillerA2.UnSuspend();
	EM_TransportFillers.UnSuspend();
	EM_OutfeedFillers.UnSuspend();
END_IF

IF fb_mem.CS.Suspend THEN
	EM_FillerA1.Suspend();
	EM_FillerA2.Suspend();
	EM_TransportFillers.Suspend();
	EM_OutfeedFillers.Suspend();
END_IF

IF fb_mem.CS.UnHold THEN
	EM_FillerA1.UnHold();
	EM_FillerA2.UnHold();
	EM_TransportFillers.UnHold();
	EM_OutfeedFillers.UnHold();
END_IF

IF fb_mem.CS.Hold THEN
	EM_FillerA1.Hold();
	EM_FillerA2.Hold();
	EM_TransportFillers.Hold();
	EM_OutfeedFillers.Hold();
END_IF

//********************************Exeptionhandling***********************************

//********************************Action case***********************************
CASE fb_mem.STS.State OF
	E_State_PackML.IDLE 			: 
		//Do nothing
	E_State_PackML.STARTING 		:
		EM_FillerA1.Start();
		IF EM_FillerA1.State 			= E_State_PackML.EXECUTE THEN
			EM_FillerA2.Start();
			IF EM_FillerA2.State 			= E_State_PackML.EXECUTE THEN
				EM_TransportFillers.Start();
				IF EM_TransportFillers.State	= E_State_PackML.EXECUTE THEN
					EM_OutfeedFillers.Start();
					IF EM_OutfeedFillers.State		= E_State_PackML.EXECUTE THEN
						fb_mem.STS.Starting_SC 		:= TRUE;
					END_IF
				END_IF
			END_IF
		END_IF
	E_State_PackML.EXECUTE 			: 
		// MAIN LOGIC:

		
	E_State_PackML.COMPLETE 		:
		IF fb_mem.CS.Clear AND fb_mem.STS.Auto OR fb_mem.HMI.Clear AND fb_mem.STS.Manueel THEN
			fb_mem.STS.Completing_SC := TRUE;
		END_IF
	E_State_PackML.RESETTING 		:
		EM_FillerA1.Reset();
		EM_FillerA2.Reset();
		EM_TransportFillers.Reset();
		EM_OutfeedFillers.Reset();
		IF 	EM_FillerA1.State 			= E_State_PackML.IDLE AND 
			EM_FillerA2.State 			= E_State_PackML.IDLE AND 
			EM_TransportFillers.State	= E_State_PackML.IDLE AND 
			EM_OutfeedFillers.State		= E_State_PackML.IDLE THEN
				fb_mem.STS.Resetting_SC 		:= TRUE;	
		END_IF
	E_State_PackML.HOLDING 			:
		EM_FillerA1.Hold();
		EM_FillerA2.Hold();
		EM_TransportFillers.Hold();
		EM_OutfeedFillers.Hold();
		IF 	EM_FillerA1.State 			= E_State_PackML.HELD AND
			EM_FillerA2.State 			= E_State_PackML.HELD AND
			EM_TransportFillers.State 	= E_State_PackML.HELD AND
			EM_OutfeedFillers.State 	= E_State_PackML.HELD THEN
				fb_mem.STS.HOLDING_SC	:= TRUE;
		END_IF
	E_State_PackML.HELD 			:
		//Do nothing
	E_State_PackML.UNHOLDING 		:
		EM_FillerA1.Unhold();
		EM_FillerA2.Unhold();
		EM_TransportFillers.Unhold();
		EM_OutfeedFillers.Unhold();
		IF 	EM_FillerA1.State 			= E_State_PackML.EXECUTE AND
			EM_FillerA2.State 			= E_State_PackML.EXECUTE AND
			EM_TransportFillers.State 	= E_State_PackML.EXECUTE AND
			EM_OutfeedFillers.State 	= E_State_PackML.EXECUTE THEN
				fb_mem.STS.UNHOLDING_SC	:= TRUE;
		END_IF;
	E_State_PackML.SUSPENDING 		:
		EM_FillerA1.Suspend();
		EM_FillerA2.Suspend();
		EM_TransportFillers.Suspend();
		EM_OutfeedFillers.Suspend();
		IF 	EM_FillerA1.State 			= E_State_PackML.SUSPENDED AND
			EM_FillerA2.State 			= E_State_PackML.SUSPENDED AND
			EM_TransportFillers.State 	= E_State_PackML.SUSPENDED AND
			EM_OutfeedFillers.State 	= E_State_PackML.SUSPENDED THEN
				fb_mem.STS.Suspending_SC	:= TRUE;
		END_IF
	E_State_PackML.SUSPENDED 		:			// TO BE PROGRAMMED
		//Do nothing
	E_State_PackML.UNSUSPENDING 	:
		EM_FillerA1.Unsuspend();
		EM_FillerA2.Unsuspend();
		EM_TransportFillers.Unsuspend();
		EM_OutfeedFillers.Unsuspend();
		IF 	EM_FillerA1.State 			= E_State_PackML.EXECUTE AND
			EM_FillerA2.State 			= E_State_PackML.EXECUTE AND
			EM_TransportFillers.State 	= E_State_PackML.EXECUTE AND
			EM_OutfeedFillers.State 	= E_State_PackML.EXECUTE THEN
				fb_mem.STS.Unsuspending_SC	:= TRUE;
		END_IF
	E_State_PackML.ABORTING			:
		EM_FillerA1.Abort();
		EM_FillerA2.Abort();
		EM_TransportFillers.Abort();
		EM_OutfeedFillers.Abort();
		IF 	EM_FillerA1.State 			= E_State_PackML.ABORTED AND
			EM_FillerA2.State 			= E_State_PackML.ABORTED AND
			EM_TransportFillers.State 	= E_State_PackML.ABORTED AND
			EM_OutfeedFillers.State 	= E_State_PackML.ABORTED THEN
				fb_mem.STS.Aborting_SC:= TRUE;
		END_IF;
	E_State_PackML.ABORTED			:
		IF fb_mem.CS.Clear AND fb_mem.STS.Auto OR fb_mem.HMI.Clear AND fb_mem.STS.Manueel THEN
			EM_FillerA1.Clear();
			EM_FillerA2.Clear();
			EM_TransportFillers.Clear();
			EM_OutfeedFillers.Clear();
		END_IF
	E_State_PackML.CLEARING 		:
		IF 	EM_FillerA1.State 			= E_State_PackML.STOPPED AND
			EM_FillerA2.State 			= E_State_PackML.STOPPED AND
			EM_TransportFillers.State 	= E_State_PackML.STOPPED AND
			EM_OutfeedFillers.State 	= E_State_PackML.STOPPED THEN
				fb_mem.STS.Clearing_SC:= TRUE;
		END_IF;
	E_State_PackML.STOPPED			:
		IF fb_mem.CS.Reset AND fb_mem.STS.Auto OR fb_mem.HMI.Reset AND fb_mem.STS.Manueel THEN
			EM_FillerA1.Reset();
			EM_FillerA2.Reset();
			EM_TransportFillers.Reset();
			EM_OutfeedFillers.Reset();
		END_IF;
	
END_CASE

//********************************HMI_Connection***********************************
fb_mem.STS.StringState     := TO_STRING(fb_mem.STS.State); 

//********************************ZEROING***********************************

fb_mem.CS.Auto            := FALSE;
fb_mem.CS.Manueel         := FALSE;
fb_mem.CS.Start           := FALSE;
fb_mem.CS.Stop            := FALSE;
fb_mem.CS.Reset           := FALSE;
fb_mem.CS.Abort           := FALSE;
fb_mem.CS.Clear           := FALSE;
fb_mem.CS.UnSuspend       := FALSE;
fb_mem.CS.Suspend         := FALSE;
fb_mem.CS.UnHold          := FALSE;
fb_mem.CS.Hold            := FALSE;

{warning 'add method implementation '}
METHOD Abort : BOOL
fb_mem.CS.Abort := TRUE;
END_METHOD

METHOD Aborting_SC : BOOL
VAR_INPUT
END_VAR
fb_mem.STS.Aborting_SC := TRUE;
END_METHOD

{warning 'add method implementation '}
METHOD Auto : BOOL
fb_mem.CS.Auto := TRUE;
Auto := fb_mem.STS.Auto;
END_METHOD

{warning 'add method implementation '}
METHOD Clear : BOOL
fb_mem.CS.Clear := TRUE;
END_METHOD

METHOD Clearing_SC : BOOL
VAR_INPUT
END_VAR
fb_mem.STS.Clearing_SC := TRUE;
END_METHOD

METHOD Completing_SC : BOOL
VAR_INPUT
END_VAR
fb_mem.STS.Completing_SC := TRUE;
END_METHOD

METHOD Execute_SC : BOOL
VAR_INPUT
END_VAR
fb_mem.STS.Execute_SC := TRUE;
END_METHOD

METHOD FB_init : BOOL
VAR_INPUT
	bInitRetains : BOOL; // if TRUE, the retain variables are initialized (warm start / cold start)
	bInCopyCode : BOOL;  // if TRUE, the instance afterwards gets moved into the copy code (online change)
END_VAR
//**************************INITIATE**************************//
END_METHOD

{warning 'add method implementation '}
METHOD Hold : BOOL
fb_mem.CS.Hold := TRUE;
END_METHOD

METHOD Holding_SC : BOOL
VAR_INPUT
END_VAR
fb_mem.STS.Holding_SC := TRUE;
END_METHOD

{warning 'add method implementation '}
METHOD Manueel : BOOL
fb_mem.CS.Manueel := TRUE;
Manueel := fb_mem.STS.Manueel;
END_METHOD

{warning 'add method implementation '}
METHOD Reset : BOOL
fb_mem.CS.Reset := TRUE;
END_METHOD

METHOD Resetting_SC : BOOL
VAR_INPUT
END_VAR
fb_mem.STS.Resetting_SC := TRUE;
END_METHOD

{warning 'add method implementation '}
METHOD Start : BOOL
fb_mem.CS.Start := TRUE;
END_METHOD

METHOD Starting_SC : BOOL
VAR_INPUT
END_VAR
fb_mem.STS.Starting_SC := TRUE;
END_METHOD

{warning 'add property implementation'}
PROPERTY State : E_State_PackML
GET
State := fb_mem.STS.State;
END_GET
END_PROPERTY

{warning 'add method implementation '}
METHOD Stop : BOOL
fb_mem.CS.Stop := TRUE;
END_METHOD

METHOD Stopping_SC : BOOL
VAR_INPUT
END_VAR
fb_mem.STS.Stopping_SC := TRUE;
END_METHOD

{warning 'add method implementation '}
METHOD Suspend : BOOL
fb_mem.CS.Suspend := TRUE;
END_METHOD

METHOD Suspending_SC : BOOL
VAR_INPUT
END_VAR
fb_mem.STS.Suspending_SC := TRUE;
END_METHOD

{warning 'add method implementation '}
METHOD Unhold : BOOL
fb_mem.CS.Unhold := TRUE;
END_METHOD

METHOD Unholding_SC : BOOL
VAR_INPUT
END_VAR
fb_mem.STS.Unholding_SC := TRUE;
END_METHOD

{warning 'add method implementation '}
METHOD Unsuspend : BOOL
fb_mem.CS.Unsuspend := TRUE;
END_METHOD

METHOD Unsuspending_SC : BOOL
VAR_INPUT
END_VAR
fb_mem.STS.Unsuspending_SC := TRUE;
END_METHOD

{warning 'add method implementation '}
METHOD ZeroAllVar : BOOL
END_METHOD

END_FUNCTION_BLOCK

// ---- POUs/2. Equipment Modules/3. EM_Machine/EM_Machine.TcPOU
FUNCTION_BLOCK EM_Machine IMPLEMENTS  ITF_PackMLV2
VAR_INPUT
END_VAR
VAR_OUTPUT
END_VAR
VAR
	fb_mem	: STRUCT_EM_Machine;
	ton1	: ton;
END_VAR

(*
$$$$$$$$\                                                                   $$\       $$$$$$$$\                     $$\                                         $$\                     
$$  _____|                                                                  $$ |      $$  _____|                    \__|                                        \__|                    
$$ |   $$$$$$\   $$$$$$\  $$$$$$$\  $$\  $$\  $$\  $$$$$$\   $$$$$$\   $$$$$$$ |      $$ |      $$$$$$$\   $$$$$$\  $$\ $$$$$$$\   $$$$$$\   $$$$$$\   $$$$$$\  $$\ $$$$$$$\   $$$$$$\  
$$$$$\ \____$$\ $$  __$$\ $$  __$$\ $$ | $$ | $$ |$$  __$$\ $$  __$$\ $$  __$$ |      $$$$$\    $$  __$$\ $$  __$$\ $$ |$$  __$$\ $$  __$$\ $$  __$$\ $$  __$$\ $$ |$$  __$$\ $$  __$$\ 
$$  __|$$$$$$$ |$$ |  \__|$$ |  $$ |$$ | $$ | $$ |$$ /  $$ |$$ /  $$ |$$ /  $$ |      $$  __|   $$ |  $$ |$$ /  $$ |$$ |$$ |  $$ |$$$$$$$$ |$$$$$$$$ |$$ |  \__|$$ |$$ |  $$ |$$ /  $$ |
$$ |  $$  __$$ |$$ |      $$ |  $$ |$$ | $$ | $$ |$$ |  $$ |$$ |  $$ |$$ |  $$ |      $$ |      $$ |  $$ |$$ |  $$ |$$ |$$ |  $$ |$$   ____|$$   ____|$$ |      $$ |$$ |  $$ |$$ |  $$ |
$$ |  \$$$$$$$ |$$ |      $$ |  $$ |\$$$$$\$$$$  |\$$$$$$  |\$$$$$$  |\$$$$$$$ |      $$$$$$$$\ $$ |  $$ |\$$$$$$$ |$$ |$$ |  $$ |\$$$$$$$\ \$$$$$$$\ $$ |      $$ |$$ |  $$ |\$$$$$$$ |
\__|   \_______|\__|      \__|  \__| \_____\____/  \______/  \______/  \_______|      \________|\__|  \__| \____$$ |\__|\__|  \__| \_______| \_______|\__|      \__|\__|  \__| \____$$ |
                                                                                                          $$\   $$ |                                                          $$\   $$ |
                                                                                                          \$$$$$$  |                                                          \$$$$$$  |
                                                                                                           \______/                                                            \______/ 
*)
//********************************Initiating***********************************
fb_mem.STS.State := PackML_StateMachine(State			:= fb_mem.STS.State,
										Start           := fb_mem.CS.Start,
										Stop            := fb_mem.CS.Stop,
										Reset           := fb_mem.CS.Reset,
										Abort           := fb_mem.CS.Abort,
										Clear           := fb_mem.CS.Clear,
										UnSuspend       := fb_mem.CS.UnSuspend,
										Suspend         := fb_mem.CS.Suspend,
										UnHold          := fb_mem.CS.UnHold,
										Hold            := fb_mem.CS.Hold,
										Starting_SC     := fb_mem.STS.Starting_SC,
										Execute_SC      := fb_mem.STS.Execute_SC,
										Completing_SC	:= fb_mem.STS.Completing_SC,
										Resetting_SC    := fb_mem.STS.Resetting_SC,
										Holding_SC      := fb_mem.STS.Holding_SC,
										Unholding_SC    := fb_mem.STS.Unholding_SC,
										Suspending_SC   := fb_mem.STS.Suspending_SC,
										Unsuspending_SC := fb_mem.STS.Unsuspending_SC,
										Aborting_SC     := fb_mem.STS.Aborting_SC,
										Clearing_SC     := fb_mem.STS.Clearing_SC,
										Stopping_SC     := fb_mem.STS.Stopping_SC);
										
//********************************ZEROING***********************************								
fb_mem.STS.Starting_SC 		:= FALSE;
fb_mem.STS.Execute_SC 		:= FALSE;
fb_mem.STS.Resetting_SC 	:= FALSE;
fb_mem.STS.Holding_SC 		:= FALSE;
fb_mem.STS.Unholding_SC 	:= FALSE;
fb_mem.STS.Suspending_SC 	:= FALSE;
fb_mem.STS.Unsuspending_SC 	:= FALSE;
fb_mem.STS.Aborting_SC 		:= FALSE;
fb_mem.STS.Clearing_SC 		:= FALSE;
fb_mem.STS.Stopping_SC 		:= FALSE;
fb_mem.STS.Completing_SC 	:= FALSE;

//********************************Auto manual logic***********************************
IF fb_mem.CS.Auto OR fb_mem.HMI.Auto THEN
	fb_mem.STS.Auto := TRUE;
	fb_mem.STS.Manueel := FALSE;
END_IF

IF fb_mem.CS.Manueel OR fb_mem.HMI.Manueel THEN
	fb_mem.STS.Auto := FALSE;
	fb_mem.STS.Manueel := TRUE;
END_IF

//********************************Action case***********************************

// THIS CODE SIMULATES A EXTERNAL MACHINE WICH RUNS ON PACKML. SO NO ACTION CASE IS PROGRAMMED


//********************************HMI_Connection***********************************
fb_mem.STS.StringState     := TO_STRING(fb_mem.STS.State); 

//********************************ZEROING***********************************

fb_mem.CS.Auto            := FALSE;
fb_mem.CS.Manueel         := FALSE;
fb_mem.CS.Start           := FALSE;
fb_mem.CS.Stop            := FALSE;
fb_mem.CS.Reset           := FALSE;
fb_mem.CS.Abort           := FALSE;
fb_mem.CS.Clear           := FALSE;
fb_mem.CS.UnSuspend       := FALSE;
fb_mem.CS.Suspend         := FALSE;
fb_mem.CS.UnHold          := FALSE;
fb_mem.CS.Hold            := FALSE;

{warning 'add method implementation '}
METHOD Abort : BOOL
fb_mem.CS.Abort := TRUE;
END_METHOD

METHOD Aborting_SC : BOOL
VAR_INPUT
END_VAR
fb_mem.STS.Aborting_SC := TRUE;
END_METHOD

{warning 'add method implementation '}
METHOD Auto : BOOL
fb_mem.CS.Auto := TRUE;
Auto := fb_mem.STS.Auto;
END_METHOD

{warning 'add method implementation '}
METHOD Clear : BOOL
fb_mem.CS.Clear := TRUE;
END_METHOD

METHOD Clearing_SC : BOOL
VAR_INPUT
END_VAR
fb_mem.STS.Clearing_SC := TRUE;
END_METHOD

METHOD Completing_SC : BOOL
VAR_INPUT
END_VAR
fb_mem.STS.Completing_SC := TRUE;
END_METHOD

METHOD Execute_SC : BOOL
VAR_INPUT
END_VAR
fb_mem.STS.Execute_SC := TRUE;
END_METHOD

METHOD FB_init : BOOL
VAR_INPUT
	bInitRetains : BOOL; // if TRUE, the retain variables are initialized (warm start / cold start)
	bInCopyCode : BOOL;  // if TRUE, the instance afterwards gets moved into the copy code (online change)
END_VAR
//**************************INITIATE**************************//
END_METHOD

{warning 'add method implementation '}
METHOD Hold : BOOL
fb_mem.CS.Hold := TRUE;
END_METHOD

METHOD Holding_SC : BOOL
VAR_INPUT
END_VAR
fb_mem.STS.Holding_SC := TRUE;
END_METHOD

{warning 'add method implementation '}
METHOD Manueel : BOOL
fb_mem.CS.Manueel := TRUE;
Manueel := fb_mem.STS.Manueel;
END_METHOD

{warning 'add method implementation '}
METHOD Reset : BOOL
fb_mem.CS.Reset := TRUE;
END_METHOD

METHOD Resetting_SC : BOOL
VAR_INPUT
END_VAR
fb_mem.STS.Resetting_SC := TRUE;
END_METHOD

{warning 'add method implementation '}
METHOD Start : BOOL
fb_mem.CS.Start := TRUE;
END_METHOD

METHOD Starting_SC : BOOL
VAR_INPUT
END_VAR
fb_mem.STS.Starting_SC := TRUE;
END_METHOD

{warning 'add property implementation'}
PROPERTY State : E_State_PackML
GET
State := fb_mem.STS.State;
END_GET
END_PROPERTY

{warning 'add method implementation '}
METHOD Stop : BOOL
fb_mem.CS.Stop := TRUE;
END_METHOD

METHOD Stopping_SC : BOOL
VAR_INPUT
END_VAR
fb_mem.STS.Stopping_SC := TRUE;
END_METHOD

{warning 'add method implementation '}
METHOD Suspend : BOOL
fb_mem.CS.Suspend := TRUE;
END_METHOD

METHOD Suspending_SC : BOOL
VAR_INPUT
END_VAR
fb_mem.STS.Suspending_SC := TRUE;
END_METHOD

{warning 'add method implementation '}
METHOD Unhold : BOOL
fb_mem.CS.Unhold := TRUE;
END_METHOD

METHOD Unholding_SC : BOOL
VAR_INPUT
END_VAR
fb_mem.STS.Unholding_SC := TRUE;
END_METHOD

{warning 'add method implementation '}
METHOD Unsuspend : BOOL
fb_mem.CS.Unsuspend := TRUE;
END_METHOD

METHOD Unsuspending_SC : BOOL
VAR_INPUT
END_VAR
fb_mem.STS.Unsuspending_SC := TRUE;
END_METHOD

{warning 'add method implementation '}
METHOD ZeroAllVar : BOOL
END_METHOD

END_FUNCTION_BLOCK

// ---- POUs/4. Management/1. AlarmHandler/AlarmHandler.TcPOU
FUNCTION_BLOCK AlarmHandler
VAR_INPUT
END_VAR
VAR_OUTPUT
END_VAR
VAR
END_VAR


VAR
	ErrorArray:ARRAY[1..3] OF stErrorHandling;
	ShowAlarms:BOOL;
END_VAR

ErrorArray[1].sTag:='Valv_StopT1';
ErrorArray[1].sMessage:= 'Temprature of motor is rising';
ErrorArray[1].sPriority:= 3;
ErrorArray[1].sDevice:= 'b_CM_Valve_CanStopper_CanSupply';
ErrorArray[1].dErrorTime:= DT#2024-2-4-14:44:44;
ErrorArray[1].sPossibleSolution:= 'Check heatsink or motor itself';
IF ErrorArray[1].bAcknowledged = 1 THEN
	ErrorArray[1].bIsAlarmAcknowledged:=1;
END_IF


ErrorArray[2].sTag:='ConveyerT1_Detect';
ErrorArray[2].sMessage:= 'Sensor is giving timeout';
ErrorArray[2].sPriority:= 2;
ErrorArray[2].sDevice:= 'ConveyerT1_Detect';
ErrorArray[2].dErrorTime:= DT#2024-2-4-14:50:44;
ErrorArray[2].sPossibleSolution:= 'Check for dust blocking the sensor or conection cable';

IF ErrorArray[2].bAcknowledged = 1 THEN
	ErrorArray[2].bIsAlarmAcknowledged:=1;
END_IF

ErrorArray[3].sTag:='Conveyer T3';
ErrorArray[3].sMessage:= 'Conveyer belt T3 is having more friction than accepted';
ErrorArray[3].sPriority:= 4;
ErrorArray[3].sDevice:= 'Conveyer Belt T3';
ErrorArray[3].dErrorTime:= DT#2024-2-4-14:59:44;
ErrorArray[3].sPossibleSolution:= 'Check the spinning friction of the belt rollers or check the motor itself.';
IF ErrorArray[3].bAcknowledged = 1 THEN
	ErrorArray[3].bIsAlarmAcknowledged:=1;
END_IF

END_FUNCTION_BLOCK

// ---- POUs/4. Management/2. ModeSelect/ModeSelect.TcPOU
FUNCTION_BLOCK ModeSelect IMPLEMENTS ITF_ModeSelect
VAR
	fb_mem : STRUCT_ModeSelect;
END_VAR

(*
$$$$$$$$\                                                                   $$\       $$$$$$$$\                     $$\                                         $$\                     
$$  _____|                                                                  $$ |      $$  _____|                    \__|                                        \__|                    
$$ |   $$$$$$\   $$$$$$\  $$$$$$$\  $$\  $$\  $$\  $$$$$$\   $$$$$$\   $$$$$$$ |      $$ |      $$$$$$$\   $$$$$$\  $$\ $$$$$$$\   $$$$$$\   $$$$$$\   $$$$$$\  $$\ $$$$$$$\   $$$$$$\  
$$$$$\ \____$$\ $$  __$$\ $$  __$$\ $$ | $$ | $$ |$$  __$$\ $$  __$$\ $$  __$$ |      $$$$$\    $$  __$$\ $$  __$$\ $$ |$$  __$$\ $$  __$$\ $$  __$$\ $$  __$$\ $$ |$$  __$$\ $$  __$$\ 
$$  __|$$$$$$$ |$$ |  \__|$$ |  $$ |$$ | $$ | $$ |$$ /  $$ |$$ /  $$ |$$ /  $$ |      $$  __|   $$ |  $$ |$$ /  $$ |$$ |$$ |  $$ |$$$$$$$$ |$$$$$$$$ |$$ |  \__|$$ |$$ |  $$ |$$ /  $$ |
$$ |  $$  __$$ |$$ |      $$ |  $$ |$$ | $$ | $$ |$$ |  $$ |$$ |  $$ |$$ |  $$ |      $$ |      $$ |  $$ |$$ |  $$ |$$ |$$ |  $$ |$$   ____|$$   ____|$$ |      $$ |$$ |  $$ |$$ |  $$ |
$$ |  \$$$$$$$ |$$ |      $$ |  $$ |\$$$$$\$$$$  |\$$$$$$  |\$$$$$$  |\$$$$$$$ |      $$$$$$$$\ $$ |  $$ |\$$$$$$$ |$$ |$$ |  $$ |\$$$$$$$\ \$$$$$$$\ $$ |      $$ |$$ |  $$ |\$$$$$$$ |
\__|   \_______|\__|      \__|  \__| \_____\____/  \______/  \______/  \_______|      \________|\__|  \__| \____$$ |\__|\__|  \__| \_______| \_______|\__|      \__|\__|  \__| \____$$ |
                                                                                                          $$\   $$ |                                                          $$\   $$ |
                                                                                                          \$$$$$$  |                                                          \$$$$$$  |
                                                                                                           \______/                                                            \______/ 
*)

{warning 'add method implementation '}
METHOD Auto : BOOL
fb_mem.Auto 	:= TRUE;
fb_mem.Manueel 	:= FALSE;

RETURN(fb_mem.Auto);
END_METHOD

{warning 'add method implementation '}
METHOD Manueel : BOOL
fb_mem.Auto 	:= FALSE;
fb_mem.Manueel 	:= TRUE;

RETURN(fb_mem.Manueel);
END_METHOD

{warning 'add property implementation'}
PROPERTY Tag : STRING
GET
Tag := fb_mem.Tag;
END_GET
SET
fb_mem.Tag := Tag;
END_SET
END_PROPERTY

END_FUNCTION_BLOCK

// ---- LIB/1. Control Modules/Brisq/1. DEV_Base/FB_DeviceBase.TcPOU
FUNCTION_BLOCK FB_DeviceBase
VAR
	TagName : STRING;
	Description : STRING;
	TagID : INT;
END_VAR

END_FUNCTION_BLOCK

// ---- LIB/1. Control Modules/Brisq/2. DEV_AnaIn/FB_DEV_AnaIn.TcPOU
FUNCTION_BLOCK FB_DEV_AnaIn EXTENDS FB_DeviceBase IMPLEMENTS ITF_DEV_AnaIn
VAR_INPUT
END_VAR
VAR_OUTPUT
END_VAR
VAR
END_VAR

END_FUNCTION_BLOCK

// ---- LIB/1. Control Modules/Brisq/3. DEV_DigIn/FB_DEV_DigIn.TcPOU
FUNCTION_BLOCK FB_DEV_DigIn EXTENDS FB_DeviceBase IMPLEMENTS ITF_DigIn
VAR
	
END_VAR

{warning 'add property implementation'}
PROPERTY ActualValue : BOOL
GET
END_GET
SET
END_SET
END_PROPERTY

{warning 'add property implementation'}
PROPERTY FallingEdge : BOOL
GET
END_GET
SET
END_SET
END_PROPERTY

{warning 'add method implementation '}
METHOD FB_init : BOOL
VAR_INPUT
	(* if TRUE, the retain variables are initialized (warm start / cold start)*)
	bInitRetains	: BOOL;
	(* if TRUE, the instance afterwards gets moved into the copy code (online change)*)
	bInCopyCode	: BOOL;
END_VAR
END_METHOD

{warning 'add method implementation '}
METHOD Force : BOOL
VAR_INPUT
	ForceValue	: BOOL;
END_VAR
END_METHOD

{warning 'add method implementation '}
METHOD ResetForce : BOOL
END_METHOD

{warning 'add property implementation'}
PROPERTY RisingEdge : BOOL
GET
END_GET
SET
END_SET
END_PROPERTY

END_FUNCTION_BLOCK

// ---- LIB/1. Control Modules/Brisq/4. DEV_Valve/DEV_Valve.TcPOU
FUNCTION_BLOCK DEV_Valve EXTENDS FB_DeviceBase IMPLEMENTS ITF_Valve

VAR
	I_FeedbackOpen		AT	%I* : BOOL;
	I_FeedbackClosed 	AT 	%I* : BOOL;
	I_Estop				AT	%I*	: BOOL;
	Q_ValveOutput		AT	%Q*	: BOOL;
	
	s_eActualState				: E_ValveState;
	s_eOperatingMode			: E_OperationMode;
	s_tonFeedbackTime			: TON;
	
	bFeedbackError		: BOOL;
	bEstopActive		: BOOL;
	bBothFeedback		: BOOL;
END_VAR

METHOD _FExceptions : BOOL
VAR_INPUT
END_VAR
END_METHOD

METHOD PRIVATE _StHmi
VAR_INPUT
	stHMI : stDevValve;
END_VAR
END_METHOD

{warning 'add property implementation'}
PROPERTY ActualState : E_ValveState
GET
END_GET
END_PROPERTY

{warning 'add method implementation '}
METHOD Close : BOOL
END_METHOD

{warning 'add property implementation'}
PROPERTY EmergencyStatus : BOOL
GET
END_GET
END_PROPERTY

{warning 'add method implementation '}
METHOD Open : BOOL
END_METHOD

{warning 'add property implementation'}
PROPERTY OperatingMode : BOOL
GET
END_GET
END_PROPERTY

{warning 'add method implementation '}
METHOD Reset : BOOL
END_METHOD

{warning 'add method implementation '}
METHOD SetMode : BOOL
END_METHOD

END_FUNCTION_BLOCK

// ---- LIB/1. Control Modules/Brisq/5. DEV_ControlValve/DEV_CtrlValve.TcPOU
FUNCTION_BLOCK DEV_CtrlValve EXTENDS FB_DeviceBase IMPLEMENTS ITF_ControlValve
VAR_INPUT
END_VAR
VAR_OUTPUT
END_VAR
VAR
END_VAR

{warning 'add property implementation'}
PROPERTY EmergencyStatus : BOOL
GET
END_GET
END_PROPERTY

{warning 'add property implementation'}
PROPERTY OperatingMode : BOOL
GET
END_GET
END_PROPERTY

{warning 'add property implementation'}
PROPERTY OutputValue : REAL
GET
END_GET
END_PROPERTY

{warning 'add method implementation '}
METHOD Reset : BOOL
END_METHOD

{warning 'add method implementation '}
METHOD SetMode : BOOL
END_METHOD

{warning 'add method implementation '}
METHOD SetValue : BOOL
END_METHOD

END_FUNCTION_BLOCK

// ---- LIB/1. Control Modules/Brisq/FB_Devices.TcPOU
FUNCTION_BLOCK FB_Devices
VAR
	devValveV2012 : DEV_Valve := (TagName := 'V2012', Description := 'Standard Valve', TagID := 1);
	devValveV2020 : DEV_Valve := (TagName := 'V2020', Description := 'Standard Valve', TagID := 2);
	devValveV2021 : DEV_Valve := (TagName := 'V2021', Description := 'Standard Valve', TagID := 3);
	devValveV2022 : DEV_Valve := (TagName := 'V2022', Description := 'Standard Valve', TagID := 4);
END_VAR

devValveV2012();
devValveV2020();
devValveV2021();
devValveV2020();

END_FUNCTION_BLOCK

// ---- LIB/2. Equipment Modules/1. FB_Base/FB_EMbase.TcPOU
FUNCTION_BLOCK FB_EMbase
VAR
	TagName : STRING;
	Description : STRING;
	TagID : INT;
END_VAR

END_FUNCTION_BLOCK

// ---- LIB/2. Equipment Modules/2. EM_Machine_PackML/FB_Machine_PackML.TcPOU
FUNCTION_BLOCK FB_Machine_PackML IMPLEMENTS ITF_PackML
VAR
	fbPackML_mem 	: STRUCT_Machine_PackML;
	StepSwitch		: E_State_PackML;
END_VAR

(*
$$$$$$$$\                                                                   $$\       $$$$$$$$\                     $$\                                         $$\                     
$$  _____|                                                                  $$ |      $$  _____|                    \__|                                        \__|                    
$$ |   $$$$$$\   $$$$$$\  $$$$$$$\  $$\  $$\  $$\  $$$$$$\   $$$$$$\   $$$$$$$ |      $$ |      $$$$$$$\   $$$$$$\  $$\ $$$$$$$\   $$$$$$\   $$$$$$\   $$$$$$\  $$\ $$$$$$$\   $$$$$$\  
$$$$$\ \____$$\ $$  __$$\ $$  __$$\ $$ | $$ | $$ |$$  __$$\ $$  __$$\ $$  __$$ |      $$$$$\    $$  __$$\ $$  __$$\ $$ |$$  __$$\ $$  __$$\ $$  __$$\ $$  __$$\ $$ |$$  __$$\ $$  __$$\ 
$$  __|$$$$$$$ |$$ |  \__|$$ |  $$ |$$ | $$ | $$ |$$ /  $$ |$$ /  $$ |$$ /  $$ |      $$  __|   $$ |  $$ |$$ /  $$ |$$ |$$ |  $$ |$$$$$$$$ |$$$$$$$$ |$$ |  \__|$$ |$$ |  $$ |$$ /  $$ |
$$ |  $$  __$$ |$$ |      $$ |  $$ |$$ | $$ | $$ |$$ |  $$ |$$ |  $$ |$$ |  $$ |      $$ |      $$ |  $$ |$$ |  $$ |$$ |$$ |  $$ |$$   ____|$$   ____|$$ |      $$ |$$ |  $$ |$$ |  $$ |
$$ |  \$$$$$$$ |$$ |      $$ |  $$ |\$$$$$\$$$$  |\$$$$$$  |\$$$$$$  |\$$$$$$$ |      $$$$$$$$\ $$ |  $$ |\$$$$$$$ |$$ |$$ |  $$ |\$$$$$$$\ \$$$$$$$\ $$ |      $$ |$$ |  $$ |\$$$$$$$ |
\__|   \_______|\__|      \__|  \__| \_____\____/  \______/  \______/  \_______|      \________|\__|  \__| \____$$ |\__|\__|  \__| \_______| \_______|\__|      \__|\__|  \__| \____$$ |
                                                                                                          $$\   $$ |                                                          $$\   $$ |
                                                                                                          \$$$$$$  |                                                          \$$$$$$  |
                                                                                                           \______/                                                            \______/ 
*)

CASE StepSwitch OF
	E_State_PackML.IDLE 			: 
		//HAPPY FLOW		
		IF fbPackML_mem.Start AND fbPackML_mem.Abort = FALSE THEN
			StepSwitch := E_State_PackML.STARTING;
		END_IF
		
		//EXEPTION HANDLING
		IF fbPackML_mem.Abort THEN
			StepSwitch:= E_State_PackML.ABORTING;
		END_IF
		IF (fbPackML_mem.Stop := TRUE) THEN
			StepSwitch:= E_State_PackML.STOPPING;
		END_IF
	
	E_State_PackML.STARTING 		:
		//HAPPY FLOW		
		IF fbPackML_mem.Starting_SC AND NOT fbPackML_mem.Abort THEN
			StepSwitch:= E_State_PackML.IDLE;
		END_IF
		
		//EXEPTION HANDLING
		IF fbPackML_mem.Abort THEN
			StepSwitch:= E_State_PackML.ABORTING;
		END_IF
		IF fbPackML_mem.Stop THEN
			StepSwitch:= E_State_PackML.STOPPING;
		END_IF
	
	E_State_PackML.EXECUTE 			: 
		//HAPPY FLOW		
		IF (fbPackML_mem.Execute_SC) AND (NOT fbPackML_mem.Abort) THEN
			StepSwitch:= E_State_PackML.IDLE;
		END_IF
		
		IF fbPackML_mem.Hold THEN
			StepSwitch:= E_State_PackML.HOLDING;
		END_IF
		
		IF fbPackML_mem.Suspend THEN
			StepSwitch := E_State_PackML.SUSPENDED;
		END_IF
		
		//EXEPTION HANDLING
		IF fbPackML_mem.Abort THEN
			StepSwitch:= E_State_PackML.ABORTING;
		END_IF
		IF fbPackML_mem.Stop THEN
			StepSwitch:= E_State_PackML.STOPPING;
		END_IF
	
	E_State_PackML.COMPLETE 		:
		//HAPPY FLOW
		StepSwitch:= E_State_PackML.RESETTING;
	
	E_State_PackML.RESETTING 		:
		//HAPPY FLOW		
		IF fbPackML_mem.Resetting_SC AND NOT fbPackML_mem.Abort THEN
			StepSwitch:= E_State_PackML.IDLE;
		END_IF
		
		//EXEPTION HANDLING
		IF fbPackML_mem.Abort THEN
			StepSwitch:= E_State_PackML.ABORTING;
		END_IF
		IF fbPackML_mem.Stop THEN
			StepSwitch:= E_State_PackML.STOPPING;
		END_IF
	
	E_State_PackML.HOLDING 			:
		//HAPPY FLOW		
		IF fbPackML_mem.Holding_SC AND NOT fbPackML_mem.Abort THEN
			StepSwitch:= E_State_PackML.HELD;
		END_IF
		
		//EXEPTION HANDLING
		IF fbPackML_mem.Abort THEN
			StepSwitch:= E_State_PackML.ABORTING;
		END_IF
		IF fbPackML_mem.Stop THEN
			StepSwitch:= E_State_PackML.STOPPING;
		END_IF
		
	
	E_State_PackML.HELD 			:
		//HAPPY FLOW		
		IF fbPackML_mem.Unhold AND NOT fbPackML_mem.Abort THEN
			StepSwitch := E_State_PackML.UNHOLDING;
		END_IF
		
		//EXEPTION HANDLING
		IF fbPackML_mem.Abort THEN
			StepSwitch:= E_State_PackML.ABORTING;
		END_IF
		IF fbPackML_mem.Stop THEN
			StepSwitch:= E_State_PackML.STOPPING;
		END_IF
	
	E_State_PackML.UNHOLDING 		:
		//HAPPY FLOW		
		IF fbPackML_mem.Unholding_SC AND NOT fbPackML_mem.Abort THEN
			StepSwitch:= E_State_PackML.EXECUTE;
		END_IF
		
		//EXEPTION HANDLING
		IF fbPackML_mem.Abort THEN
			StepSwitch:= E_State_PackML.ABORTING;
		END_IF
		IF fbPackML_mem.Stop THEN
			StepSwitch:= E_State_PackML.STOPPING;
		END_IF
	
	E_State_PackML.SUSPENDING 		:
		//HAPPY FLOW		
		IF fbPackML_mem.Suspending_SC AND NOT fbPackML_mem.Abort THEN
			StepSwitch:= E_State_PackML.SUSPENDED;
		END_IF
		
		//EXEPTION HANDLING
		IF fbPackML_mem.Abort THEN
			StepSwitch:= E_State_PackML.ABORTING;
		END_IF
		IF fbPackML_mem.Stop THEN
			StepSwitch:= E_State_PackML.STOPPING;
		END_IF
	
	
	E_State_PackML.SUSPENDED 		:
		//HAPPY FLOW		
		IF fbPackML_mem.Unsuspend AND NOT fbPackML_mem.Abort THEN
			StepSwitch:= E_State_PackML.UNSUSPENDING;
		END_IF
		
		//EXEPTION HANDLING
		IF fbPackML_mem.Abort THEN
			StepSwitch:= E_State_PackML.ABORTING;
		END_IF
		IF fbPackML_mem.Stop THEN
			StepSwitch:= E_State_PackML.STOPPING;
		END_IF
	
	E_State_PackML.UNSUSPENDING 	:
		//HAPPY FLOW		
		IF fbPackML_mem.Unsuspending_SC AND NOT fbPackML_mem.Abort THEN
			StepSwitch:= E_State_PackML.EXECUTE;
		END_IF
		
		//EXEPTION HANDLING
		IF fbPackML_mem.Abort THEN
			StepSwitch:= E_State_PackML.ABORTING;
		END_IF
		IF fbPackML_mem.Stop THEN
			StepSwitch:= E_State_PackML.STOPPING;
		END_IF
	
	E_State_PackML.ABORTED			:
		//HAPPY FLOW		
		IF fbPackML_mem.Clear THEN
			StepSwitch:= E_State_PackML.CLEARING;
		END_IF
	
		
	E_State_PackML.ABORTING			:
		//HAPPY FLOW		
		IF fbPackML_mem.Aborting_SC THEN
			StepSwitch:= E_State_PackML.ABORTED;
		END_IF
	
		
	E_State_PackML.CLEARING 		:
		//HAPPY FLOW		
		IF fbPackML_mem.Clearing_SC THEN
			StepSwitch:= E_State_PackML.STOPPED;
		END_IF
		
		//EXEPTION HANDLING
		IF fbPackML_mem.Abort THEN
			StepSwitch:= E_State_PackML.ABORTING;
		END_IF
		
		
	E_State_PackML.STOPPING 		:
		//HAPPY FLOW
		IF fbPackML_mem.Stopping_SC THEN
			StepSwitch:= E_State_PackML.STOPPED;
		END_IF
		
		//EXEPTION HANDLING
		IF fbPackML_mem.Abort THEN
			StepSwitch:= E_State_PackML.ABORTING;
		END_IF
		
	
	E_State_PackML.STOPPED 			: 
		//HAPPY FLOW
		IF fbPackML_mem.Reset AND NOT fbPackML_mem.Abort THEN
			StepSwitch:= E_State_PackML.RESETTING;
		END_IF
		
		//EXEPTION HANDLING
		IF fbPackML_mem.Abort THEN
			StepSwitch:= E_State_PackML.ABORTING;
		END_IF
		IF fbPackML_mem.Stop THEN
			StepSwitch:= E_State_PackML.STOPPING;
		END_IF
END_CASE

// Set variables FALSE
(*
fbPackML_mem.Abort 			:= FALSE;
fbPackML_mem.Aborting_SC 	:= FALSE;
fbPackML_mem.Clear 			:= FALSE;
fbPackML_mem.Clearing_SC 	:= FALSE;
fbPackML_mem.Execute_SC 	:= FALSE;
fbPackML_mem.Completing_SC	:= FALSE;
fbPackML_mem.Hold 			:= FALSE;
fbPackML_mem.Holding_SC 	:= FALSE;
fbPackML_mem.Reset 			:= FALSE;
fbPackML_mem.Resetting_SC 	:= FALSE;
fbPackML_mem.Start 			:= FALSE;
fbPackML_mem.Starting_SC 	:= FALSE;
fbPackML_mem.Stop 			:= FALSE;
fbPackML_mem.Stopping_SC 	:= FALSE;
fbPackML_mem.Suspend 		:= FALSE;
fbPackML_mem.Suspending_SC 	:= FALSE;
fbPackML_mem.Unhold 		:= FALSE;
fbPackML_mem.Unholding_SC 	:= FALSE;
fbPackML_mem.Unsuspend 		:= FALSE;
*)

{warning 'add method implementation '}
METHOD Abort : BOOL
fbPackML_mem.Abort := TRUE;
END_METHOD

{warning 'add method implementation '}
METHOD Aborting_SC : BOOL
fbPackML_mem.Aborting_SC := TRUE;
END_METHOD

{warning 'add method implementation '}
METHOD Clear : BOOL
fbPackML_mem.Clear := TRUE;
END_METHOD

{warning 'add method implementation '}
METHOD Clearing_SC : BOOL
fbPackML_mem.Clearing_SC := TRUE;
END_METHOD

{warning 'add method implementation '}
METHOD Completing_SC : BOOL
fbPackML_mem.Completing_SC := TRUE;
END_METHOD

{warning 'add method implementation '}
METHOD Execute_SC : BOOL
fbPackML_mem.Execute_SC := TRUE;
END_METHOD

{warning 'add method implementation '}
METHOD FB_init : BOOL
VAR_INPUT
	(* if TRUE, the retain variables are initialized (warm start / cold start)*)
	bInitRetains	: BOOL;
	(* if TRUE, the instance afterwards gets moved into the copy code (online change)*)
	bInCopyCode	: BOOL;
END_VAR
END_METHOD

{warning 'add method implementation '}
METHOD Hold : BOOL
fbPackML_mem.Hold := TRUE;
END_METHOD

{warning 'add method implementation '}
METHOD Holding_SC : BOOL
fbPackML_mem.Holding_SC := TRUE;
END_METHOD

{warning 'add method implementation '}
METHOD Reset : BOOL
fbPackML_mem.Reset := TRUE;
END_METHOD

{warning 'add method implementation '}
METHOD Resetting_SC : BOOL
fbPackML_mem.Resetting_SC := TRUE;
END_METHOD

{warning 'add method implementation '}
METHOD Start : BOOL
fbPackML_mem.Start := TRUE;
END_METHOD

{warning 'add method implementation '}
METHOD Starting_SC : BOOL
fbPackML_mem.Starting_SC := TRUE;
END_METHOD

{warning 'add property implementation'}
PROPERTY State : E_State_PackML
GET
State := StepSwitch;
END_GET
END_PROPERTY

{warning 'add method implementation '}
METHOD Stop : BOOL
fbPackML_mem.Stop := TRUE;
END_METHOD

{warning 'add method implementation '}
METHOD Stopping_SC : BOOL
fbPackML_mem.Stopping_SC := TRUE;
END_METHOD

{warning 'add method implementation '}
METHOD Suspend : BOOL
fbPackML_mem.Suspend := TRUE;
END_METHOD

{warning 'add method implementation '}
METHOD Suspending_SC : BOOL
fbPackML_mem.Suspending_SC := TRUE;
END_METHOD

{warning 'add method implementation '}
METHOD Unhold : BOOL
fbPackML_mem.Unhold := TRUE;
END_METHOD

{warning 'add method implementation '}
METHOD Unholding_SC : BOOL
fbPackML_mem.Unholding_SC := TRUE;
END_METHOD

{warning 'add method implementation '}
METHOD Unsuspend : BOOL
fbPackML_mem.Unsuspend := TRUE;
END_METHOD

METHOD Unsuspending_SC : BOOL
VAR_INPUT
END_VAR
fbPackML_mem.Unsuspending_SC := TRUE;
END_METHOD

{warning 'add method implementation '}
METHOD ZeroAllVar : BOOL
END_METHOD

END_FUNCTION_BLOCK

// ---- LIB/3. Units/1. UN_Base/FB_UN_base.TcPOU
FUNCTION_BLOCK FB_UN_base
VAR
	TagName : STRING;
	Description : STRING;
	TagID : INT;
END_VAR

END_FUNCTION_BLOCK
